Omron CX-Programmer project NuevoProyecto (CX-Programmer 9.54)

# PLC NuevoPLC1: CQM1 CPU41

## Program NuevoPrograma1 (no task)
Local symbols
ET0 20.04 BOOL
ET1 20.05 BOOL
ET10 20.14 BOOL
ET11 20.15 BOOL
ET2 20.06 BOOL
ET3 20.07 BOOL
ET4 20.08 BOOL
ET5 20.09 BOOL
ET6 20.10 BOOL
ET7 20.11 BOOL
ET8 20.12 BOOL
ET9 20.13 BOOL
FBS2 20.00 BOOL  ; FLANCO BAJADA SENSOR 2
FBS4 20.01 BOOL  ; FLANCO BAJADA SENSOR 4
FCIIN 0.14 BOOL
FCIOUT 0.15 BOOL
FCSIN 0.06 BOOL
FCSOUT 0.07 BOOL
H_1 100.11 BOOL
H_2 100.03 BOOL
IGU10 20.02 BOOL  ; IGUAL A 10
M1B 100.08 BOOL
M1S 100.00 BOOL
M2B 100.15 BOOL
M2S 100.07 BOOL
MEN10 20.03 BOOL  ; MENOR 10
PM 0.00 BOOL  ; PULSADOR MARCHA
PP 0.01 BOOL  ; PULSADOR PARO
RESET 0.03 BOOL  ; RSET DEL SISTEMA
SE1 0.04 BOOL
SE2 0.05 BOOL
SE3 0.08 BOOL
SE4 0.09 BOOL
SE5 0.02 BOOL

### Section PROG_PRINC

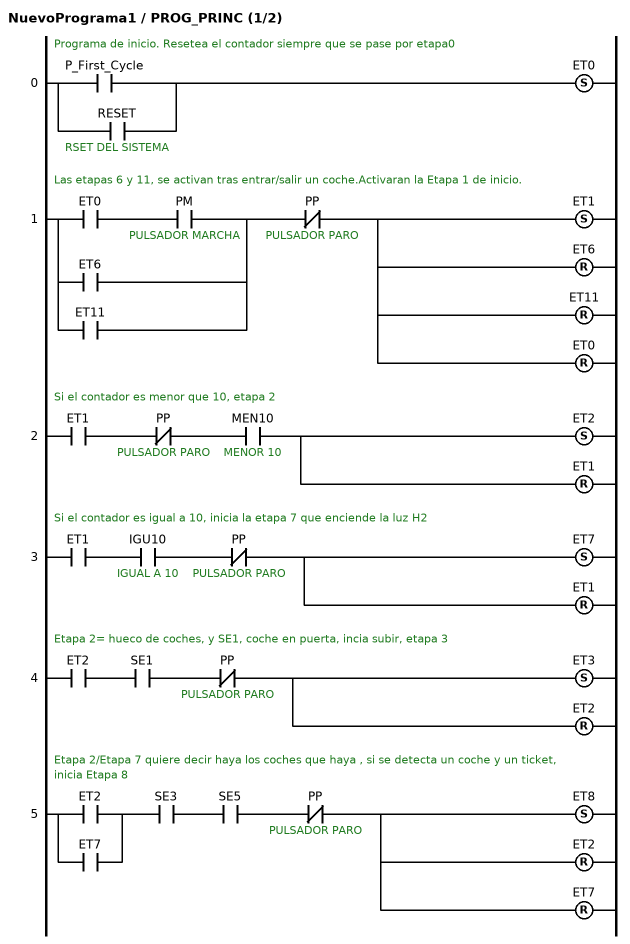
; rung 0: Programa de inicio. Resetea el contador siempre que se pase por etapa0
LD P_First_Cycle
OR RESET  ; RSET DEL SISTEMA
SET ET0
; rung 1: Las etapas 6 y 11, se activan tras entrar/salir un coche.Activaran la Etapa 1 de inicio.
LD ET0
AND PM  ; PULSADOR MARCHA
OR ET6
OR ET11
ANDNOT PP  ; PULSADOR PARO
SET ET1
RSET ET6
RSET ET11
RSET ET0
; rung 2: Si el contador es menor que 10, etapa 2
LD ET1
ANDNOT PP  ; PULSADOR PARO
AND MEN10  ; MENOR 10
SET ET2
RSET ET1
; rung 3: Si el contador es igual a 10, inicia la etapa 7 que enciende la luz H2
LD ET1
AND IGU10  ; IGUAL A 10
ANDNOT PP  ; PULSADOR PARO
SET ET7
RSET ET1
; rung 4: Etapa 2= hueco de coches, y SE1, coche en puerta, incia subir, etapa 3
LD ET2
AND SE1
ANDNOT PP  ; PULSADOR PARO
SET ET3
RSET ET2
; rung 5: Etapa 2/Etapa 7 quiere decir haya los coches que haya , si se detecta un coche y un ticket, inicia Etapa 8
LD ET2
OR ET7
AND SE3
AND SE5
ANDNOT PP  ; PULSADOR PARO
SET ET8
RSET ET2
RSET ET7

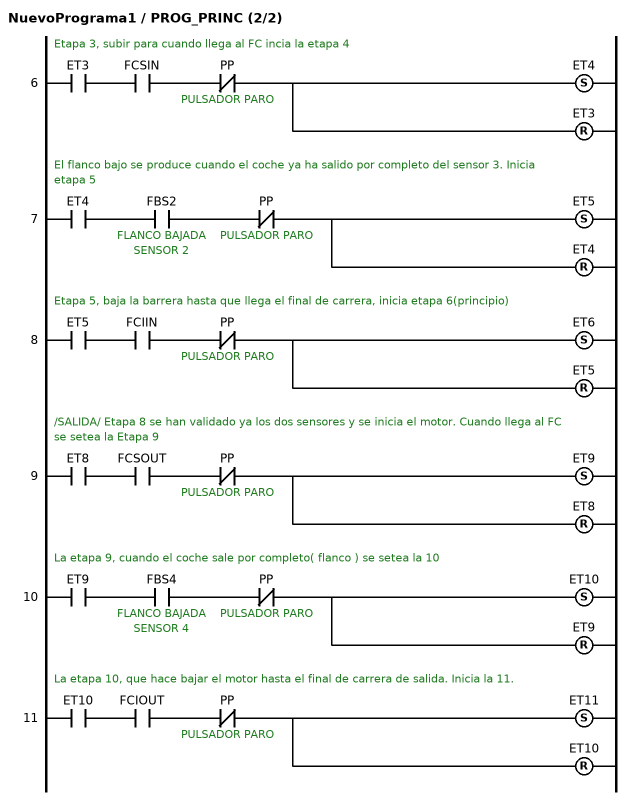
; rung 6: Etapa 3, subir para cuando llega al FC incia la etapa 4
LD ET3
AND FCSIN
ANDNOT PP  ; PULSADOR PARO
SET ET4
RSET ET3
; rung 7: El flanco bajo se produce cuando el coche ya ha salido por completo del sensor 3. Inicia etapa 5
LD ET4
AND FBS2  ; FLANCO BAJADA SENSOR 2
ANDNOT PP  ; PULSADOR PARO
SET ET5
RSET ET4
; rung 8: Etapa 5, baja la barrera hasta que llega el final de carrera, inicia etapa 6(principio)
LD ET5
AND FCIIN
ANDNOT PP  ; PULSADOR PARO
SET ET6
RSET ET5
; rung 9: /SALIDA/ Etapa 8 se han validado ya los dos sensores y se inicia el motor. Cuando llega al FC se setea la Etapa 9
LD ET8
AND FCSOUT
ANDNOT PP  ; PULSADOR PARO
SET ET9
RSET ET8
; rung 10: La etapa 9, cuando el coche sale por completo( flanco ) se setea la 10
LD ET9
AND FBS4  ; FLANCO BAJADA SENSOR 4
ANDNOT PP  ; PULSADOR PARO
SET ET10
RSET ET9
; rung 11: La etapa 10, que hace bajar el motor hasta el final de carrera de salida. Inicia la 11.
LD ET10
AND FCIOUT
ANDNOT PP  ; PULSADOR PARO
SET ET11
RSET ET10

### Section ETAPAS

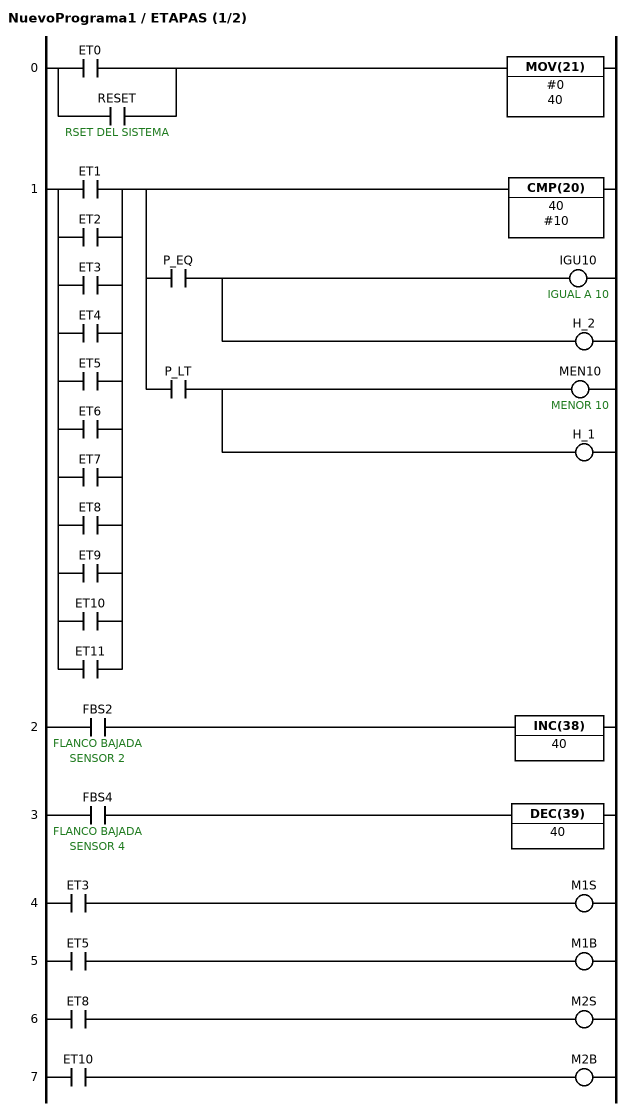
; rung 0
LD ET0
OR RESET  ; RSET DEL SISTEMA
MOV(21) #0 40
; rung 1
LD ET1
OR ET2
OR ET3
OR ET4
OR ET5
OR ET6
OR ET7
OR ET8
OR ET9
OR ET10
OR ET11
OUT TR0
CMP(20) 40 #10
AND P_EQ
OUT IGU10  ; IGUAL A 10
OUT H_2
LD TR0
AND P_LT
OUT MEN10  ; MENOR 10
OUT H_1
; rung 2
LD FBS2  ; FLANCO BAJADA SENSOR 2
INC(38) 40
; rung 3
LD FBS4  ; FLANCO BAJADA SENSOR 4
DEC(39) 40
; rung 4
LD ET3
OUT M1S
; rung 5
LD ET5
OUT M1B
; rung 6
LD ET8
OUT M2S
; rung 7
LD ET10
OUT M2B

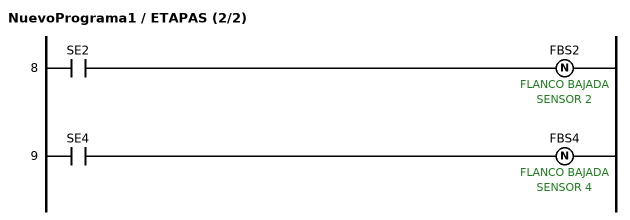
; rung 8
LD SE2
DIFD(14) FBS2  ; FLANCO BAJADA SENSOR 2
; rung 9
LD SE4
DIFD(14) FBS4  ; FLANCO BAJADA SENSOR 4

### Section END
; rung 0
END(01)